{attribute addProperty BoxType "AX8206-0000-0102-0102"}
{attribute addProperty Id "DeviceDevice_F82A60211620Ch_ACh_A_B17182A2176220Ch_BCh_B_7239D878176220WcStateAT %I*WcState_F855686C1620InfoDataAT %I*InfoData_17277C5A208260"}
{attribute addProperty CRC "1305851277"}
{attribute addProperty SizeInBites "592"}
{attribute addProperty SizeInBytes "74"}
TYPE AX8206_DA6659A9 :
STRUCT
	{attribute addProperty Name "Device"}
	Device : Device_F82A6021;
	{attribute addProperty Name "Ch_A"}
	Ch_A : Ch_A_B17182A2;
	{attribute addProperty Name "Ch_B"}
	Ch_B : Ch_B_7239D878;
	{attribute addProperty Name "WcState"}
	WcState : WcState_F855686C;
	{attribute addProperty Name "InfoData"}
	InfoData : InfoData_17277C5A;
END_STRUCT
END_TYPE

(* stored: Version 1.2.0.0, ProductVersion 3.1.4024.9
   DUT AX8206_DA6659A9: Id {3a512f2f-50df-4d47-b2b5-9340326d36b6} *)
